SUBAPPLICATION mapping_Softkeys (* Subapplication Type *)
  (* Standard: 61499-2 *)
  (* Version 1.0, 2023-01-29, Franz *)
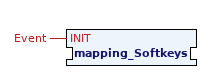
  EVENT_INPUT
    INIT;
  END_EVENT
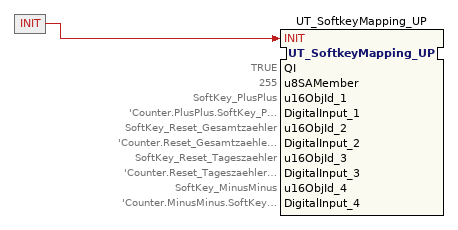
  FBS
    UT_SoftkeyMapping_UP : UT_SoftkeyMapping_UP(QI := TRUE, u8SAMember := 255, u16ObjId_1 := SoftKey_PlusPlus, DigitalInput_1 := 'Counter.PlusPlus.SoftKey_PlusPlus', u16ObjId_2 := SoftKey_Reset_Gesamtzaehler, DigitalInput_2 := 'Counter.Reset_Gesamtzaehler.SoftKey_Reset_Gesamtzaehler', u16ObjId_3 := SoftKey_Reset_Tageszaehler, DigitalInput_3 := 'Counter.Reset_Tageszaehler.SoftKey_Reset_Tageszaehler', u16ObjId_4 := SoftKey_MinusMinus, DigitalInput_4 := 'Counter.MinusMinus.SoftKey_MinusMinus');
  END_FBS
  EVENT_CONNECTIONS
    INIT TO UT_SoftkeyMapping_UP.INIT;
  END_CONNECTIONS
END_SUBAPPLICATION
